FUNCTION_BLOCK FB_Sensor_NC
VAR_INPUT
END_VAR
VAR_OUTPUT
END_VAR
VAR
END_VAR

END_FUNCTION_BLOCK

(* stored: Version 1.1.0.1, ProductVersion 3.1.4024.12
   POU FB_Sensor_NC: Id {f26a07d0-e6ea-484e-8faf-33c29b957afa}, SpecialFunc None *)
